VAR_GLOBAL
    (*
      PD33 series laser displacement sensor (Modbus RTU over EL6022 / RS-485).

      Registers (from manual screenshots):
      Current mode: passive parsing of PD33 full-speed active output.
      Expected frame: slave=1, function=3, bytecount=4, payload i32 low-word-first, CRC16.
      Scale: raw / 1000.0 = mm.
    *)

    Enable : BOOL;
    Channel : USINT := 1; // 1 or 2 (EL6022 channel)
    SlaveId : USINT := 1; // Modbus address

    // PD33 frames shown in the manual interpret 32-bit values as "low word first".
    // Keep this TRUE unless you verify your device uses the opposite order.
    WordSwap32 : BOOL := TRUE;
    UseDisplayRegister3B : BOOL := FALSE; // reserved; passive full-speed output parser does not send read requests

    // Command handshake (PC writes Cmd+CmdSeq; PLC sets CmdAckSeq after completion)
    CmdSeq : UDINT;
    Cmd : USINT; // reserved in passive mode
    CmdAckSeq : UDINT;
    Busy : BOOL;

    // Diagnostics
    ChannelConflict : BOOL; // TRUE when another driver is using the same EL6022 channel
    PortReady : BOOL;
    CommOk : BOOL;
    CommErrorCount : UDINT;
    LastErrorId : UDINT;
    ExceptionCode : USINT;
    RxDiscardCount : UDINT;
    LastDiscardId : UDINT;

    // Measurements
    AbsRaw : DINT; // raw units depend on UseDisplayRegister3B
    RelRaw : DINT; // raw units depend on UseDisplayRegister3B
    AbsMm : LREAL; // computed
    RelMm : LREAL; // computed

    ZeroWord : UINT; // last written value to 0x0020 (for debug)

    // Debug frames (last Modbus tx/rx)
    LastTxLen : USINT;
    LastTx : ARRAY [0..21] OF USINT;
    LastRxLen : USINT;
    LastRx : ARRAY [0..21] OF USINT;
END_VAR

(* stored: Version 1.1.0.1, ProductVersion 3.1.4024.13
   GVL GVL_PD33: Id {0c1e2c71-0f0b-4a16-9d21-7a52be7c4f9b} *)
